(* CODESYS project SmiuUGP.project

Project tree, tasks and I/O mapping:
  CODESYS_Control_for_Raspberry_Pi : CODESYS Control for Raspberry Pi, 3S - Smart Software Solutions GmbH, version 3.5.7.10
    application Application
      libraries: Util, * (System)
      task MainTask (cyclic, interval t#4ms, priority 1) calls PLC_PRG, GPIO_HANDLER
      task VISU_TASK (cyclic, interval 100 ms, priority 30) calls VisuElems.Visu_Prg
      program PLC_PRG [CFC]
      visualisation test
      visualisation Visualization_Bplus
      program GPIO_HANDLER [ST]
    SoftMotion General Axis Pool
    GPIOs_B_Pi2 : GPIOs B+/Pi2, 3S - Smart Software Solutions GmbH, version 1.1.1.10
        input  Application.GPIO_HANDLER.IN_10 : BOOL  // digital inputs (GPIO0..GPIO31).Bit5
        input  Application.GPIO_HANDLER.IN_12 : BOOL  // digital inputs (GPIO0..GPIO31).Bit6
        input  Application.GPIO_HANDLER.IN_9 : BOOL  // digital inputs (GPIO0..GPIO31).Bit7
        input  Application.GPIO_HANDLER.IN_8 : BOOL  // digital inputs (GPIO0..GPIO31).Bit8
        input  Application.GPIO_HANDLER.IN_3 : BOOL  // digital inputs (GPIO0..GPIO31).Bit10
        input  Application.GPIO_HANDLER.IN_11 : BOOL  // digital inputs (GPIO0..GPIO31).Bit12
        input  Application.GPIO_HANDLER.IN_1 : BOOL  // digital inputs (GPIO0..GPIO31).Bit13
        input  Application.GPIO_HANDLER.IN_6 : BOOL  // digital inputs (GPIO0..GPIO31).Bit18
        input  Application.GPIO_HANDLER.IN_7 : BOOL  // digital inputs (GPIO0..GPIO31).Bit21
        input  Application.GPIO_HANDLER.IN_5 : BOOL  // digital inputs (GPIO0..GPIO31).Bit23
        input  Application.GPIO_HANDLER.IN_4 : BOOL  // digital inputs (GPIO0..GPIO31).Bit24
        input  Application.GPIO_HANDLER.IN_2 : BOOL  // digital inputs (GPIO0..GPIO31).Bit25
        unmapped channels: digital inputs (GPIO0..GPIO31), digital outputs (GPIO0..GPIO31)
    Camera device
      <Empty>
    I²C
    SPI
    Onewire
    Ethernet : Ethernet, 3S - Smart Software Solutions GmbH, version 3.4.2.0
        settings: IPAddress = [192,168,10,190]; SubnetMask = [255,255,255,0]; GatewayAddress = [192,168,10,1]; NetworkInterfaceName = "ether0"
      Modbus_TCP_Master : Modbus TCP Master, 3S - Smart Software Solutions GmbH, version 3.5.4.0
          settings: AutoReconnect = TRUE
        IPS_1 : Modbus TCP Slave, 3S - Smart Software Solutions GmbH, version 3.5.4.0
            settings: Unit-ID = 1; ResponseTimeout = 1500; IPAddress = [192, 168, 10, 189]; Input_group.Function Code = 3; Input_group.Read Offset = 16#000B; Input_group.Read Length = 20; Input_group.Write Offset = 0; Input_group.Write Length = 0; Input_group.Cycle Time = 300
            unmapped channels: Input_group
    Modbus_COM : Modbus COM, 3S - Smart Software Solutions GmbH, version 3.4.0.0
        settings: DataBits = 8; StopBits = 1; ComPort = 1
      Modbus_Master_COM_Port : Modbus Master, COM Port, 3S - Smart Software Solutions GmbH, version 3.5.5.0
          settings: Transmission = 'RTU'; ResponseTimeout = 1000; TimeBetweenFrames = 10; Auto-restart communication = TRUE
        MV110 : Modbus Slave, COM Port, 3S - Smart Software Solutions GmbH, version 3.5.4.0
            settings: SlaveAddress = 2; ResponseTimeout = 1000; UseExtendedFunctionCodes = TRUE; Channel 0.Function Code = 3; Channel 0.Read Offset = 16#0001; Channel 0.Read Length = 3; Channel 0.Write Offset = 0; Channel 0.Write Length = 0; Channel 0.Cycle Time = 100
            unmapped channels: Channel 0
    Modbus_COM_1 : Modbus COM, 3S - Smart Software Solutions GmbH, version 3.4.0.0
        settings: DataBits = 8; StopBits = 1; ComPort = 2
      Modbus_Master_COM_Port_1 : Modbus Master, COM Port, 3S - Smart Software Solutions GmbH, version 3.5.5.0
          settings: Transmission = 'RTU'; ResponseTimeout = 1000; TimeBetweenFrames = 10; Auto-restart communication = TRUE
        MV110_1 : Modbus Slave, COM Port, 3S - Smart Software Solutions GmbH, version 3.5.4.0
            settings: SlaveAddress = 2; ResponseTimeout = 1000; UseExtendedFunctionCodes = TRUE; Channel 0.Function Code = 3; Channel 0.Read Offset = 16#0001; Channel 0.Read Length = 3; Channel 0.Write Offset = 0; Channel 0.Write Length = 0; Channel 0.Cycle Time = 100
            unmapped channels: Channel 0
  text list GlobalTextList
*)

// CODESYS_Control_for_Raspberry_Pi/Application/PLC_PRG
PROGRAM PLC_PRG
VAR

END_VAR

END_PROGRAM

// CODESYS_Control_for_Raspberry_Pi/Application/GPIO_HANDLER
PROGRAM GPIO_HANDLER
VAR
	IN_1: BOOL;
	IN_2: BOOL;
	IN_3: BOOL;
	IN_4: BOOL;
	IN_5: BOOL;
	IN_6: BOOL;
	IN_7: BOOL;
	IN_8: BOOL;
	IN_9: BOOL;
	IN_10: BOOL;
	IN_11: BOOL;
	IN_12: BOOL;
END_VAR

IN_1 := NOT(IN_1);
IN_2 := NOT(IN_2);
IN_3 := NOT(IN_3);
IN_4 := NOT(IN_4);
IN_5 := NOT(IN_5);
IN_6 := NOT(IN_6);
IN_7 := NOT(IN_7);
IN_8 := NOT(IN_8);
IN_9 := NOT(IN_9);
IN_10 := NOT(IN_10);
IN_11 := NOT(IN_11);
IN_12 := NOT(IN_12);

END_PROGRAM

// CODESYS_Control_for_Raspberry_Pi/Application/test
VISUALIZATION test  // 2x2
END_VISUALIZATION

// CODESYS_Control_for_Raspberry_Pi/Application/Visualization_Bplus
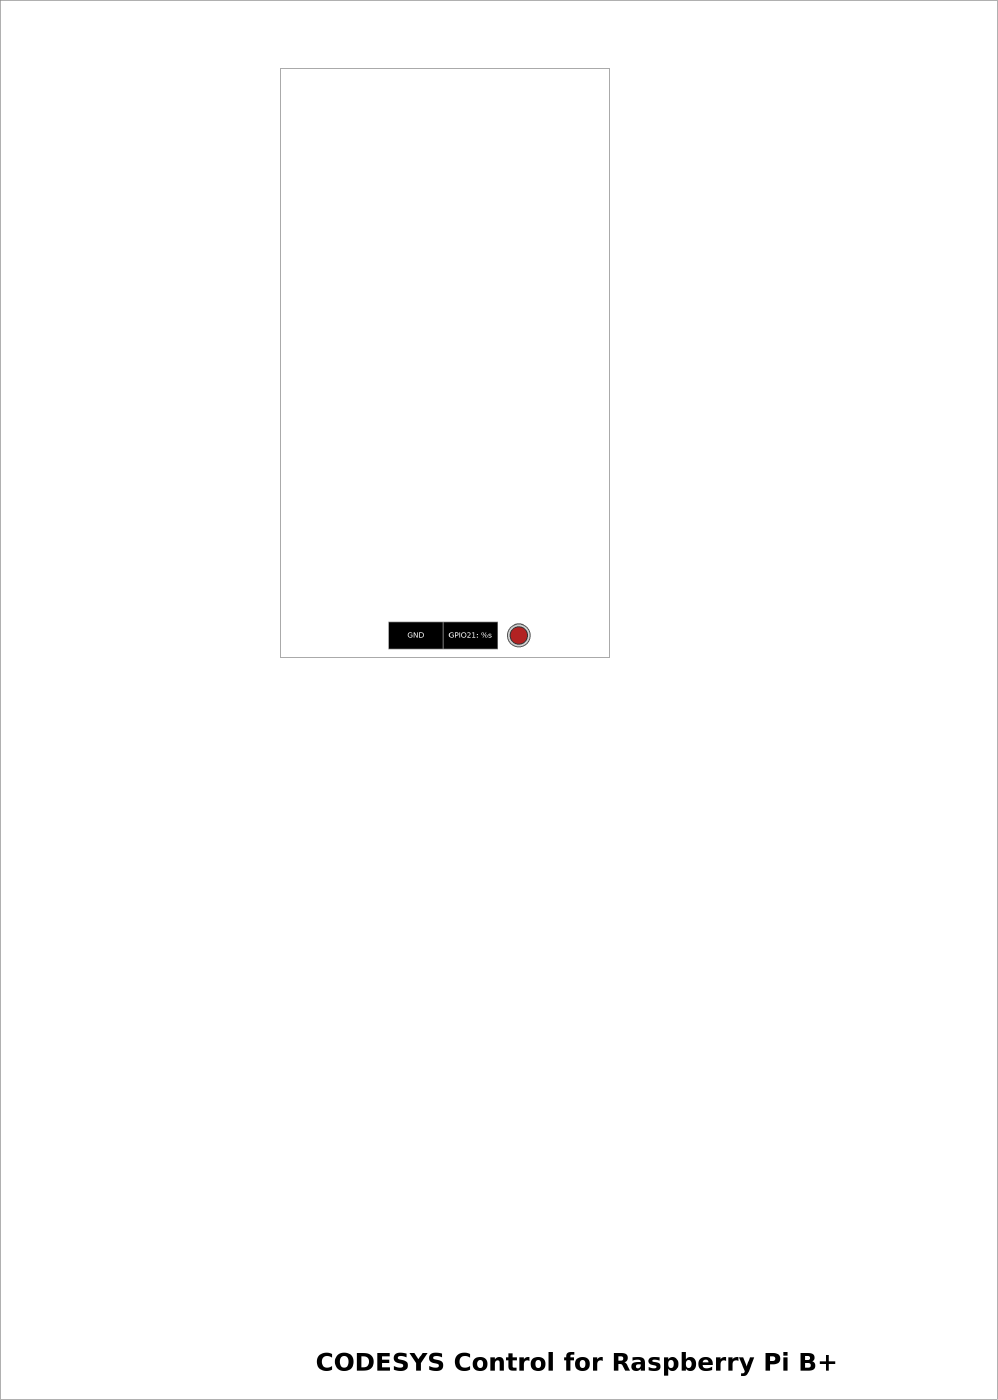
VISUALIZATION Visualization_Bplus  // 1462x2049
    Label (230,1940 1230x107), "CODESYS Control for Raspberry Pi B+"
    RoundedRectangle (410,100 483x862)
    Rectangle (649,910 80x40), "GPIO21: %s", text variable: GPIOs_Instance._GPIO.aeType[21]
    Rectangle (569,910 80x40), "GND"
    Lamp1 (740,910 40x40), variable: GPIOs_Instance._GPIO.axInputs[21], style: Lamp-Lamp1-Red
END_VISUALIZATION
